PROGRAM MAIN
VAR
	
newVar : BOOL;
END_VAR

newVar := 1;

END_PROGRAM

(* stored: Version 1.1.0.1, ProductVersion 3.1.4024.9
   POU MAIN: Id {319b139c-1377-4d52-94c4-4dd8285f8fc5}, SpecialFunc None *)
